// TIA Portal V16 export
// export: Created 2021-11-12T13:31:52.0118192Z, ExportSetting WithDefaults, DisplayName Totally Integrated Automation Portal, DisplayVersion V16 Update 3, DisplayName TIA Portal Version Control Interface, DisplayVersion V16 Update 2, DisplayName TIA Portal Openness, DisplayVersion V16 Update 3, DisplayName SINAMICS Startdrive Advanced, DisplayVersion V16 Update 5, DisplayName SINAMICS Startdrive G130, G150, S120, S150, SINAMICS MV, S210, DisplayVersion V16 Update 5, DisplayName SINAMICS Startdrive G110M, G120, G120C, G120D, G120P, G115D, DisplayVersion V16 Update 5, DisplayName STEP 7 Professional, DisplayVersion V16 Update 3, DisplayName STEP 7 Safety, DisplayVersion V16, DisplayName WinCC UA Professional, DisplayVersion V16 Update 3
DATA_BLOCK "IDB_Cab_000+UH01"   // DB14
VERSION : 0.1
// stored: AutoNumber true, DBAccessibleFromOPCUA true, InstanceOfName Cab_000+UH01, InstanceOfType FB
"Cab_000+UH01"
   // VAR
   //    SF_FV0111_Alarm { S7_SetPoint := 'True'} : "STD_DI_Mon";
   //    SF_FC0114_Alarm { S7_SetPoint := 'True'} : "STD_DI_Mon";
   //    SF_FB0114_Alarm { S7_SetPoint := 'True'} : "STD_DI_Mon";
   //    "SF_I100.3_Alarm" { S7_SetPoint := 'True'} : "STD_DI_Mon";
   //    "SF_I100.4_Alarm" { S7_SetPoint := 'True'} : "STD_DI_Mon";
   //    "SF_I100.5_Alarm" { S7_SetPoint := 'True'} : "STD_DI_Mon";
   //    "SF_I100.6_Alarm" { S7_SetPoint := 'True'} : "STD_DI_Mon";
   //    "SF_I100.7_Alarm" { S7_SetPoint := 'True'} : "STD_DI_Mon";
   //    SF_FC2114_Alarm { S7_SetPoint := 'True'} : "STD_DI_Mon";
   //    SF_EC0114_Alarm { S7_SetPoint := 'True'} : "STD_DI_Mon";
   //    SF_FC2214_Alarm { S7_SetPoint := 'True'} : "STD_DI_Mon";
   //    SF_FC2314_Alarm { S7_SetPoint := 'True'} : "STD_DI_Mon";
   //    SF_FC2414_Alarm { S7_SetPoint := 'True'} : "STD_DI_Mon";
   //    SF_FC2114_Alarm_1 { S7_SetPoint := 'True'} : "STD_DI_Mon";
   //    SF_FC2214_Alarm_1 { S7_SetPoint := 'True'} : "STD_DI_Mon";
   //    "SF_I101.7_Alarm" { S7_SetPoint := 'True'} : "STD_DI_Mon";
   //    SF_FC3014_Alarm { S7_SetPoint := 'True'} : "STD_DI_Mon";
   //    SF_FC3024_Alarm { S7_SetPoint := 'True'} : "STD_DI_Mon";
   //    SF_RB0124_Alarm { S7_SetPoint := 'True'} : "STD_DI_Mon";
   //    SF_FC5014_Alarm { S7_SetPoint := 'True'} : "STD_DI_Mon";
   //    SF_FC5024_Alarm { S7_SetPoint := 'True'} : "STD_DI_Mon";
   //    "SF_I102.5_Alarm" { S7_SetPoint := 'True'} : "STD_DI_Mon";
   //    "SF_I102.6_Alarm" { S7_SetPoint := 'True'} : "STD_DI_Mon";
   //    "SF_I102.7_Alarm" { S7_SetPoint := 'True'} : "STD_DI_Mon";
   // END_VAR
BEGIN
END_DATA_BLOCK
